INTERFACE I_CollectionDisposedEvent EXTENDS I_Event

PROPERTY PUBLIC Target : I_Collection
GET
END_GET
END_PROPERTY

END_INTERFACE

(* stored: Version 1.1.0.1, ProductVersion 3.1.4024.12
   Itf I_CollectionDisposedEvent: Id {5b531013-4022-02c6-3785-aade53ace514}
   Property Target: Id {0d2019f0-0ffa-0aea-2e02-7d20cd828742}
   Get Get: Id {e41e2ec4-176e-091f-0573-5dd4772e1bef} *)
